// SIMATIC S7-200 project (STEP 7-Micro/WIN), CPU 224XP REL 02.01

SYMBOL_TABLE USER1
start            I0.0     // khoi  dong he thong
stopp            I0.1     // dung he thong
reset            I0.2     // dat lai he thong
TLB1             I0.3     // cam bien muc nuoc tren
TLB2             I0.4     // cam bien muc nuoc duoi
MV1              Q0.0     // van 1
MV2              Q0.1     // van 2
M                Q0.2     // mo dong co
PL               Q0.3     // den bao
BZ               Q0.4     // coi bao
END_SYMBOL_TABLE

ORGANIZATION_BLOCK MAIN:OB1
TITLE=PROGRAM COMMENTS
BEGIN
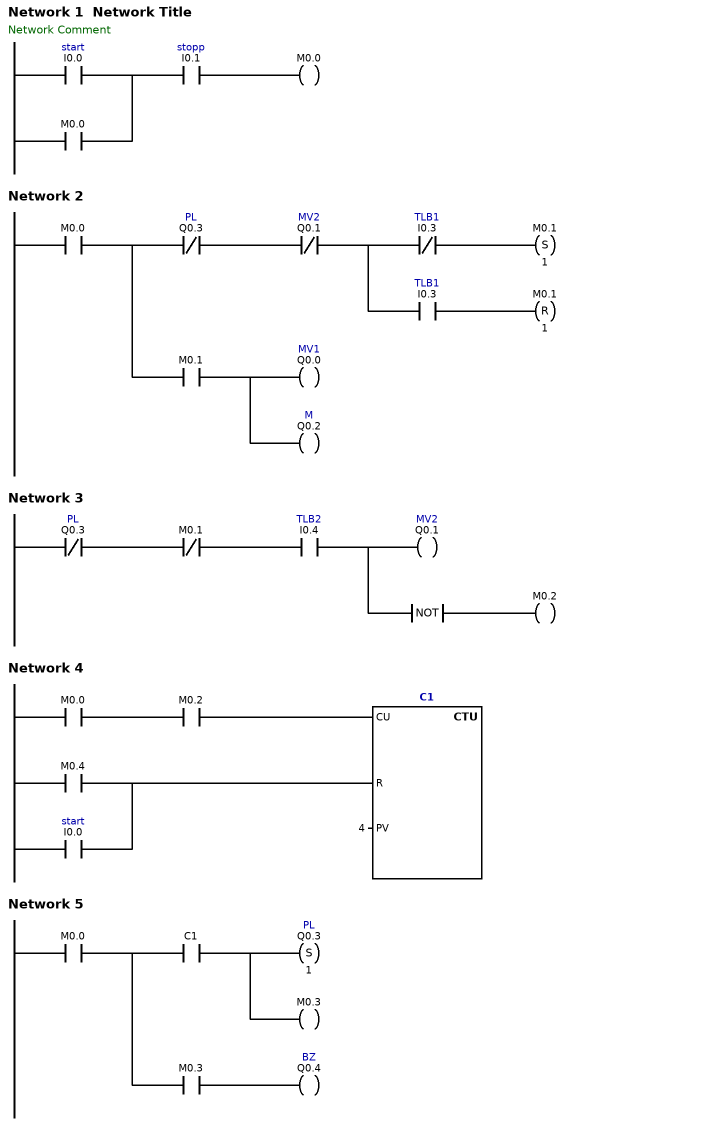
Network 1 // Network Title
// Network Comment
LD     start:I0.0
O      M0.0
A      stopp:I0.1
=      M0.0
Network 2
LD     M0.0
LPS
AN     PL:Q0.3
AN     MV2:Q0.1
LPS
AN     TLB1:I0.3
S      M0.1, 1
LPP
A      TLB1:I0.3
R      M0.1, 1
LPP
A      M0.1
=      MV1:Q0.0
=      M:Q0.2
Network 3
LDN    PL:Q0.3
AN     M0.1
A      TLB2:I0.4
=      MV2:Q0.1
NOT
=      M0.2
Network 4
LD     M0.0
A      M0.2
LD     M0.4
O      start:I0.0
CTU    C1, 4
Network 5
LD     M0.0
LPS
A      C1
S      PL:Q0.3, 1
=      M0.3
LPP
A      M0.3
=      BZ:Q0.4
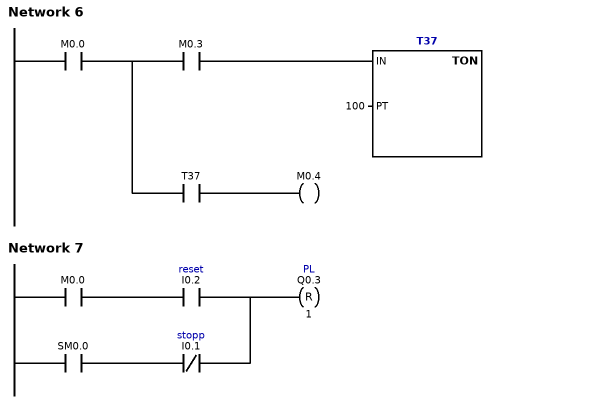
Network 6
LD     M0.0
LPS
A      M0.3
TON    T37, 100
LPP
A      T37
=      M0.4
Network 7
LD     M0.0
A      reset:I0.2
LD     SM0.0
AN     stopp:I0.1
OLD
R      PL:Q0.3, 1
END_ORGANIZATION_BLOCK
